FUNCTION_BLOCK IncrementVar
VAR
END_VAR

METHOD Increment : INT
VAR
	nValue	: INT := 5;
END_VAR
nValue := nValue + 1;
Increment := nValue;
END_METHOD

END_FUNCTION_BLOCK

(* stored: Version 1.1.0.1
   POU IncrementVar: Id {da8658d0-6e26-4098-819f-1e4637226e5b}, SpecialFunc None
   Method Increment: Id {17de9d10-e199-43cc-9c20-8df16a04ad84} *)
